ABB RobotStudio station: Project1_local_rebe.rsstnx

Station Project1_local_rebe (saved by RobotStudio 25.1.11133.0)
Controller Controlador1
  mechanical unit ROB_1: IRB120_3_58__01, 6 joints, base frame (0, 0, 0) mm
Layout (positions relative to the parent item):
  - IRB120_3_58__01 [mechanism, from %ABB.RobotStudio.Models.IRB120%\IRB120_3_58_G_01.rslib] at (0, 0, 0) mm; joint values [-0.0506, 0.4132, -0.715, -0.0948, 1.1452, -0.0907] (rad or m)
  - Herramienta_piramidal [mechanism, from Components\Herramienta_piramidal.rslib] at (0, 0, 0) mm
  - Herramienta_de_soldadura [mechanism, from Components\Herramienta_de_soldadura.rslib] at (422.9, -27.65, 640.37) mm, rotated rx -168.58 ry 40.71 rz -173.1 deg
Attachment: Herramienta_de_soldadura is attached to IRB120_3_58__01 / Link6
Targets, tools, work objects and paths stored in the station, written as RAPID:
! task T_ROB1
MODULE CalibData
  PERS tooldata Herramienta_piramidal:=[TRUE,[[0,0,160],[1,0,0,0]],[0.2,[0,0,36.89],[1,0,0,0],0,0,0]];
  PERS tooldata attach_cylinder:=[TRUE,[[0,0,0],[1,0,0,0]],[1,[-61.183,0.797,1],[1,0,0,0],0,0,0]];
  PERS tooldata puncture_figure:=[TRUE,[[-115.458,0.883,185],[1,0,0,0]],[1,[-61.183,0.797,1],[1,0,0,0],0,0,0]];
ENDMODULE

